// TIA Portal V18 export
// export: Created 2026-06-05T07:40:25.465053Z, ExportSetting WithDefaults, DisplayName Totally Integrated Automation Portal, DisplayVersion V18, DisplayName TIA Portal Openness, DisplayVersion V18, DisplayName TIA Portal Version Control Interface, DisplayVersion V18, DisplayName STEP 7 Professional, DisplayVersion V18, DisplayName STEP 7 Safety, DisplayVersion V18, DisplayName WinCC Professional, DisplayVersion V18
FUNCTION "FC_PLC2_Logic" : Void   // FC10, LAD
{ S7_Optimized_Access := 'TRUE' }
VERSION : 0.1
// stored: AutoNumber true, IsIECCheckEnabled false, SetENOAutomatically false, UDAEnableTagReadback false
BEGIN

REGION Network 1: Freq Scale: SP x 10
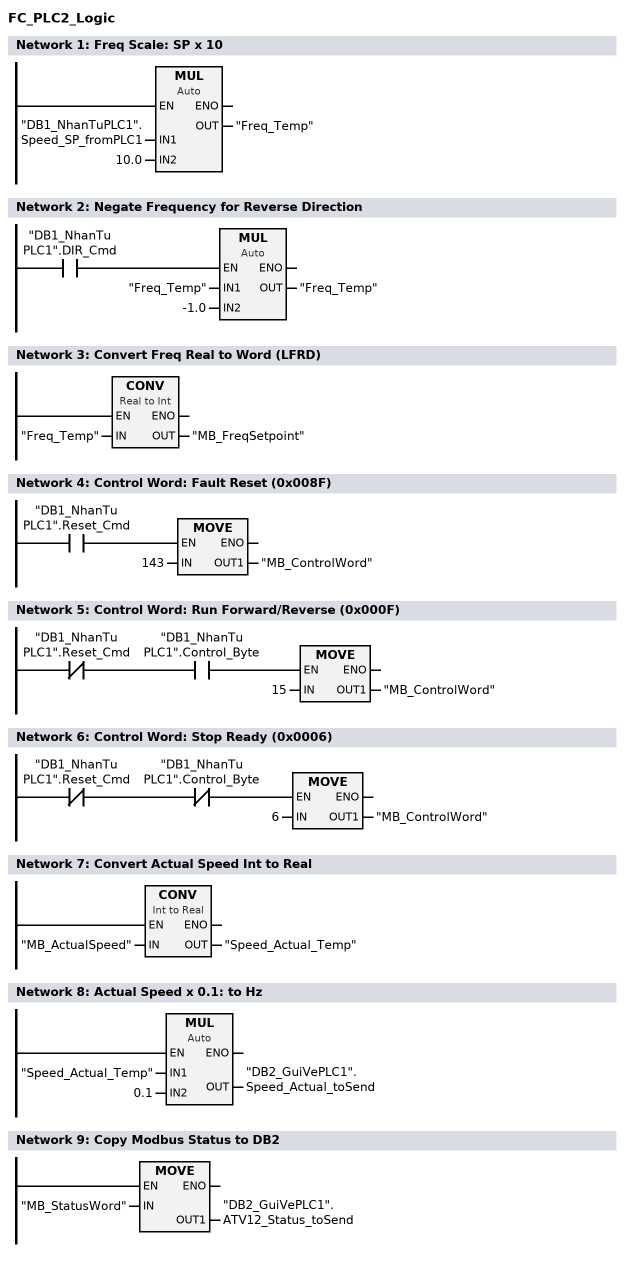
   RUNG wire#powerrail
      { S7_GenerateENO := "TRUE" } Mul(in1 := "DB1_NhanTuPLC1".Speed_SP_fromPLC1, in2 := 10.0, out => "Freq_Temp")
   END_RUNG
   // the same network as SCL:
   "Freq_Temp" := "DB1_NhanTuPLC1".Speed_SP_fromPLC1 * 10.0;
END_REGION

REGION Network 2: Negate Frequency for Reverse Direction
   RUNG wire#powerrail
      Contact( "DB1_NhanTuPLC1".DIR_Cmd )
      { S7_GenerateENO := "TRUE" } Mul(in1 := "Freq_Temp", in2 := -1.0, out => "Freq_Temp")
   END_RUNG
   // the same network as SCL:
   IF "DB1_NhanTuPLC1".DIR_Cmd THEN "Freq_Temp" := "Freq_Temp" * (-1.0); END_IF;
END_REGION

REGION Network 3: Convert Freq Real to Word (LFRD)
   RUNG wire#powerrail
      { S7_Templates := "[SrcType := Real, DestType := Int]"; S7_GenerateENO := "TRUE" } Convert(in := "Freq_Temp", out => "MB_FreqSetpoint")
   END_RUNG
   // the same network as SCL:
   "MB_FreqSetpoint" := REAL_TO_INT("Freq_Temp");
END_REGION

REGION Network 4: Control Word: Fault Reset (0x008F)
   RUNG wire#powerrail
      Contact( "DB1_NhanTuPLC1".Reset_Cmd )
      { S7_GenerateENO := "TRUE" } Move(in := 143, out1 => "MB_ControlWord")
   END_RUNG
   // the same network as SCL:
   IF "DB1_NhanTuPLC1".Reset_Cmd THEN "MB_ControlWord" := 143; END_IF;
END_REGION

REGION Network 5: Control Word: Run Forward/Reverse (0x000F)
   RUNG wire#powerrail
      I_Contact( "DB1_NhanTuPLC1".Reset_Cmd )
      Contact( "DB1_NhanTuPLC1".Control_Byte )
      { S7_GenerateENO := "TRUE" } Move(in := 15, out1 => "MB_ControlWord")
   END_RUNG
   // the same network as SCL:
   IF NOT "DB1_NhanTuPLC1".Reset_Cmd AND "DB1_NhanTuPLC1".Control_Byte THEN "MB_ControlWord" := 15; END_IF;
END_REGION

REGION Network 6: Control Word: Stop Ready (0x0006)
   RUNG wire#powerrail
      I_Contact( "DB1_NhanTuPLC1".Reset_Cmd )
      I_Contact( "DB1_NhanTuPLC1".Control_Byte )
      { S7_GenerateENO := "TRUE" } Move(in := 6, out1 => "MB_ControlWord")
   END_RUNG
   // the same network as SCL:
   IF NOT "DB1_NhanTuPLC1".Reset_Cmd AND NOT "DB1_NhanTuPLC1".Control_Byte THEN
       "MB_ControlWord" := 6;
   END_IF;
END_REGION

REGION Network 7: Convert Actual Speed Int to Real
   RUNG wire#powerrail
      { S7_Templates := "[SrcType := Int, DestType := Real]"; S7_GenerateENO := "TRUE" } Convert(in := "MB_ActualSpeed", out => "Speed_Actual_Temp")
   END_RUNG
   // the same network as SCL:
   "Speed_Actual_Temp" := INT_TO_REAL("MB_ActualSpeed");
END_REGION

REGION Network 8: Actual Speed x 0.1: to Hz
   RUNG wire#powerrail
      { S7_GenerateENO := "TRUE" } Mul(in1 := "Speed_Actual_Temp", in2 := 0.1, out => "DB2_GuiVePLC1".Speed_Actual_toSend)
   END_RUNG
   // the same network as SCL:
   "DB2_GuiVePLC1".Speed_Actual_toSend := "Speed_Actual_Temp" * 0.1;
END_REGION

REGION Network 9: Copy Modbus Status to DB2
   RUNG wire#powerrail
      { S7_GenerateENO := "TRUE" } Move(in := "MB_StatusWord", out1 => "DB2_GuiVePLC1".ATV12_Status_toSend)
   END_RUNG
   // the same network as SCL:
   "DB2_GuiVePLC1".ATV12_Status_toSend := "MB_StatusWord";
END_REGION
END_FUNCTION
